// TwinCAT 3 PLC project PLC
// ProgramVersion: 3.1.4023.0
// libraries:
//   Tc2_Standard, * (Beckhoff Automation GmbH)
//   Tc2_System, * (Beckhoff Automation GmbH)
//   Tc3_Module, * (Beckhoff Automation GmbH)
//   VisuSymbols,3.5.10.0,System
// project tree:
//   / GlobalTextList.TcGTLO, PlcTask.TcTTO, Visualization Manager.TcVMO (not stored)
//   GVLs/ Inputs.TcGVL, Outputs.TcGVL, Process.TcGVL
//   POUs/ IIRFilter.TcPOU, UpdateInterlockAndLimit.TcPOU, WriteToInterlockAndLimit.TcPOU, ByteArrayToDINT.TcPOU, ByteArrayToReal.TcPOU, CAN_Receive.TcPOU, CAN_Send.TcPOU, DINTToByteArray.TcPOU, MAIN.TcPOU, RealToByteArray.TcPOU, ScalingIn.TcPOU, ScalingOut.TcPOU
//   VISUs/ Visualization.TcVIS
// real-time tasks:
//   TASK PlcTask: cycle T#2ms, priority 20, ADS port 350
// motion (NC):
//   TASK NC-Task 1 SAF: cycle T#2ms, priority 4, ADS port 501
//   TASK NC-Task 1 SVB: cycle T#2ms, priority 8, ADS port 511
//   AXIS Axis 1 (id 1)
//     OtherSettings: AllowMotionCmdToSlave=true
//     encoder EncType=4
//       EncPara: MaxCount=#x0000ffff
//         Inc: RefSoftSyncMask=#x0000ffff
//     drive DrvType=24
//       Analog: TorqueSetpointScale=10, ScaleFactorActTorque=0.1
//       TimeComp: TaskDelayCycles=1
//     controller CtrType=1
//       CtrPara: PriorControlFactor=1
//         Observer: BandWidth=20
//   AXIS Axis 2 (id 2)
//     OtherSettings: AllowMotionCmdToSlave=true
//     encoder EncType=4
//       EncPara: ScaleFactorNumerator=0.000624, MaxCount=#x0000ffff
//         Inc: RefSoftSyncMask=#x0000ffff
//     drive DrvType=24
//       Analog: TorqueSetpointScale=10, ScaleFactorActTorque=0.1
//       TimeComp: TaskDelayCycles=1
//     controller CtrType=1
//       CtrPara: PriorControlFactor=1
//         Observer: BandWidth=20
//   AXIS Axis 3 (id 3)
//     OtherSettings: AllowMotionCmdToSlave=true
//     encoder EncType=4
//       EncPara: MaxCount=#x0000ffff
//         Inc: RefSoftSyncMask=#x0000ffff
//     drive DrvType=24
//       Analog: TorqueSetpointScale=10, ScaleFactorActTorque=0.1
//       TimeComp: TaskDelayCycles=1
//     controller CtrType=1
//       CtrPara: PriorControlFactor=1
//         Observer: BandWidth=20
//   AXIS Axis 4 (id 4)
//     OtherSettings: AllowMotionCmdToSlave=true
//     encoder EncType=4
//       EncPara: MaxCount=#x0000ffff
//         Inc: RefSoftSyncMask=#x0000ffff
//     drive DrvType=24
//       Analog: TorqueSetpointScale=10, ScaleFactorActTorque=0.1
//       TimeComp: TaskDelayCycles=1
//     controller CtrType=1
//       CtrPara: PriorControlFactor=1
//         Observer: BandWidth=20
// I/O:
//   DEVICE Device 1 (EtherCAT), AmsNetId 5.89.199.32.2.1
//     Term 1 (EK1200) [EK1200-5000 EtherCAT Power supply (2A E-Bus)]
//       Term 2 (EL2008) [EL2008 8Ch. Dig. Output 24V, 0.5A]
//       Term 3 (EL3174) [EL3174 4Ch. Ana. Input +/-10V Diff., +/-20mA SingleEnded, 16 Bit]
//       Term 4 (EL1008) [EL1008 8Ch. Dig. Input 24V, 3ms]
//       Term 6 (EL4132) [EL4132 2Ch. Ana. Output +/-10V, 16bit]
//       Term 7 (EL4132) [EL4132 2Ch. Ana. Output +/-10V, 16bit]
//       Term 8 (EL6751) [EL6751 CANopen Master]
//       Term 9 (EK1110) [EK1110 EtherCAT extension]
//     Term 10 (EK1100) [EK1100 EtherCAT Coupler (2A E-Bus)]
//       Term 11 (EL7031) [EL7031 1Ch. Stepper motor output stage (24V, 1.5A)]
//       Term 12 (EL7031) [EL7031 1Ch. Stepper motor output stage (24V, 1.5A)]
//       Term 13 (EL7031) [EL7031 1Ch. Stepper motor output stage (24V, 1.5A)]
//       Term 14 (EL7031) [EL7031 1Ch. Stepper motor output stage (24V, 1.5A)]
//       Term 15 (EL1008) [EL1008 8Ch. Dig. Input 24V, 3ms]
//       Term 16 (EL3174) [EL3174 4Ch. Ana. Input +/-10V Diff., +/-20mA SingleEnded, 16 Bit]
//       Term 17 (EL3356-0010) [EL3356-0010 1Ch. Ana. Input Resistor Bridge Terminal, 24bit, High Precision]
//       Term 18 (EL3356-0010) [EL3356-0010 1Ch. Ana. Input Resistor Bridge Terminal, 24bit, High Precision]
//       Term 19 (EL3356-0010) [EL3356-0010 1Ch. Ana. Input Resistor Bridge Terminal, 24bit, High Precision]
//       Term 5 (EL4112) [EL4112 2Ch. Ana. Output  0-20mA, 16bit]
//       Term 20 (EL9011) [EL9011 End Terminal]
//   DEVICE Device 2 (EL6751), AmsNetId 5.89.199.32.3.1
//     Box 21 (CAN Interface)
// variable links:
//   NC-Task 1 SAF/Axes/Axis 1 <-> Device 1 (EtherCAT)/Term 10 (EK1100)/Term 11 (EL7031)
//     Drive/Inputs/In/nState1 @bit 3 <-> STM Status/Status/Error
//     Drive/Inputs/In/nState1 @bit 5 <-> STM Status/Status/Moving negative
//     Drive/Inputs/In/nState1 @bit 4 <-> STM Status/Status/Moving positive
//     Drive/Inputs/In/nState1 @bit 1 <-> STM Status/Status/Ready
//     Drive/Inputs/In/nState1 <-> STM Status/Status/Ready to enable
//     Drive/Inputs/In/nState1 @bit 6 <-> STM Status/Status/Torque reduced
//     Drive/Inputs/In/nState1 @bit 2 <-> STM Status/Status/Warning
//     Drive/Inputs/In/nState2 @bit 3 <-> STM Status/Status/Digital input 1
//     Drive/Inputs/In/nState2 @bit 4 <-> STM Status/Status/Digital input 2
//     Drive/Inputs/In/nState2 @bit 5 <-> STM Status/Status/Sync error
//     Drive/Inputs/In/nState2 @bit 7 <-> STM Status/Status/TxPDO Toggle
//     Drive/Inputs/In/nState4 @bit 1 <-> WcState/InputToggle
//     Drive/Inputs/In/nState4 <-> WcState/WcState
//     Drive/Outputs/Out/nCtrl1 <-> STM Control/Control/Enable
//     Drive/Outputs/Out/nCtrl1 @bit 2 <-> STM Control/Control/Reduce torque
//     Drive/Outputs/Out/nCtrl1 @bit 1 <-> STM Control/Control/Reset
//     Drive/Outputs/Out/nDataOut2[0] <-> STM Velocity/Velocity
//     Enc/Inputs/In/nDataIn1[0] <-> ENC Status compact/Counter value
//     Enc/Inputs/In/nDataIn2[0] <-> ENC Status compact/Latch value
//     Enc/Inputs/In/nState1 @bit 4 <-> ENC Status compact/Status/Counter overflow
//     Enc/Inputs/In/nState1 @bit 3 <-> ENC Status compact/Status/Counter underflow
//     Enc/Inputs/In/nState1 @bit 1 <-> ENC Status compact/Status/Latch extern valid
//     Enc/Inputs/In/nState1 @bit 2 <-> ENC Status compact/Status/Set counter done
//     Enc/Inputs/In/nState2 @bit 4 <-> ENC Status compact/Status/Status of extern latch
//     Enc/Inputs/In/nState2 @bit 5 <-> ENC Status compact/Status/Sync error
//     Enc/Inputs/In/nState2 @bit 7 <-> ENC Status compact/Status/TxPDO Toggle
//     Enc/Inputs/In/nState4 @bit 1 <-> WcState/InputToggle
//     Enc/Inputs/In/nState4 <-> WcState/WcState
//     Enc/Outputs/Out/nCtrl1 @bit 3 <-> ENC Control compact/Control/Enable latch extern on negative edge
//     Enc/Outputs/Out/nCtrl1 @bit 1 <-> ENC Control compact/Control/Enable latch extern on positive edge
//     Enc/Outputs/Out/nCtrl1 @bit 2 <-> ENC Control compact/Control/Set counter
//     Enc/Outputs/Out/nDataOut1[0] <-> ENC Control compact/Set counter value
//   NC-Task 1 SAF/Axes/Axis 2 <-> Device 1 (EtherCAT)/Term 10 (EK1100)/Term 12 (EL7031)
//     Drive/Inputs/In/nState1 @bit 3 <-> STM Status/Status/Error
//     Drive/Inputs/In/nState1 @bit 5 <-> STM Status/Status/Moving negative
//     Drive/Inputs/In/nState1 @bit 4 <-> STM Status/Status/Moving positive
//     Drive/Inputs/In/nState1 @bit 1 <-> STM Status/Status/Ready
//     Drive/Inputs/In/nState1 <-> STM Status/Status/Ready to enable
//     Drive/Inputs/In/nState1 @bit 6 <-> STM Status/Status/Torque reduced
//     Drive/Inputs/In/nState1 @bit 2 <-> STM Status/Status/Warning
//     Drive/Inputs/In/nState2 @bit 3 <-> STM Status/Status/Digital input 1
//     Drive/Inputs/In/nState2 @bit 4 <-> STM Status/Status/Digital input 2
//     Drive/Inputs/In/nState2 @bit 5 <-> STM Status/Status/Sync error
//     Drive/Inputs/In/nState2 @bit 7 <-> STM Status/Status/TxPDO Toggle
//     Drive/Inputs/In/nState4 @bit 1 <-> WcState/InputToggle
//     Drive/Inputs/In/nState4 <-> WcState/WcState
//     Drive/Outputs/Out/nCtrl1 <-> STM Control/Control/Enable
//     Drive/Outputs/Out/nCtrl1 @bit 2 <-> STM Control/Control/Reduce torque
//     Drive/Outputs/Out/nCtrl1 @bit 1 <-> STM Control/Control/Reset
//     Drive/Outputs/Out/nDataOut2[0] <-> STM Velocity/Velocity
//     Enc/Inputs/In/nDataIn1[0] <-> ENC Status compact/Counter value
//     Enc/Inputs/In/nDataIn2[0] <-> ENC Status compact/Latch value
//     Enc/Inputs/In/nState1 @bit 4 <-> ENC Status compact/Status/Counter overflow
//     Enc/Inputs/In/nState1 @bit 3 <-> ENC Status compact/Status/Counter underflow
//     Enc/Inputs/In/nState1 @bit 1 <-> ENC Status compact/Status/Latch extern valid
//     Enc/Inputs/In/nState1 @bit 2 <-> ENC Status compact/Status/Set counter done
//     Enc/Inputs/In/nState2 @bit 4 <-> ENC Status compact/Status/Status of extern latch
//     Enc/Inputs/In/nState2 @bit 5 <-> ENC Status compact/Status/Sync error
//     Enc/Inputs/In/nState2 @bit 7 <-> ENC Status compact/Status/TxPDO Toggle
//     Enc/Inputs/In/nState4 @bit 1 <-> WcState/InputToggle
//     Enc/Inputs/In/nState4 <-> WcState/WcState
//     Enc/Outputs/Out/nCtrl1 @bit 3 <-> ENC Control compact/Control/Enable latch extern on negative edge
//     Enc/Outputs/Out/nCtrl1 @bit 1 <-> ENC Control compact/Control/Enable latch extern on positive edge
//     Enc/Outputs/Out/nCtrl1 @bit 2 <-> ENC Control compact/Control/Set counter
//     Enc/Outputs/Out/nDataOut1[0] <-> ENC Control compact/Set counter value
//   NC-Task 1 SAF/Axes/Axis 3 <-> Device 1 (EtherCAT)/Term 10 (EK1100)/Term 13 (EL7031)
//     Drive/Inputs/In/nState1 @bit 3 <-> STM Status/Status/Error
//     Drive/Inputs/In/nState1 @bit 5 <-> STM Status/Status/Moving negative
//     Drive/Inputs/In/nState1 @bit 4 <-> STM Status/Status/Moving positive
//     Drive/Inputs/In/nState1 @bit 1 <-> STM Status/Status/Ready
//     Drive/Inputs/In/nState1 <-> STM Status/Status/Ready to enable
//     Drive/Inputs/In/nState1 @bit 6 <-> STM Status/Status/Torque reduced
//     Drive/Inputs/In/nState1 @bit 2 <-> STM Status/Status/Warning
//     Drive/Inputs/In/nState2 @bit 3 <-> STM Status/Status/Digital input 1
//     Drive/Inputs/In/nState2 @bit 4 <-> STM Status/Status/Digital input 2
//     Drive/Inputs/In/nState2 @bit 5 <-> STM Status/Status/Sync error
//     Drive/Inputs/In/nState2 @bit 7 <-> STM Status/Status/TxPDO Toggle
//     Drive/Inputs/In/nState4 @bit 1 <-> WcState/InputToggle
//     Drive/Inputs/In/nState4 <-> WcState/WcState
//     Drive/Outputs/Out/nCtrl1 <-> STM Control/Control/Enable
//     Drive/Outputs/Out/nCtrl1 @bit 2 <-> STM Control/Control/Reduce torque
//     Drive/Outputs/Out/nCtrl1 @bit 1 <-> STM Control/Control/Reset
//     Drive/Outputs/Out/nDataOut2[0] <-> STM Velocity/Velocity
//     Enc/Inputs/In/nDataIn1[0] <-> ENC Status compact/Counter value
//     Enc/Inputs/In/nDataIn2[0] <-> ENC Status compact/Latch value
//     Enc/Inputs/In/nState1 @bit 4 <-> ENC Status compact/Status/Counter overflow
//     Enc/Inputs/In/nState1 @bit 3 <-> ENC Status compact/Status/Counter underflow
//     Enc/Inputs/In/nState1 @bit 1 <-> ENC Status compact/Status/Latch extern valid
//     Enc/Inputs/In/nState1 @bit 2 <-> ENC Status compact/Status/Set counter done
//     Enc/Inputs/In/nState2 @bit 4 <-> ENC Status compact/Status/Status of extern latch
//     Enc/Inputs/In/nState2 @bit 5 <-> ENC Status compact/Status/Sync error
//     Enc/Inputs/In/nState2 @bit 7 <-> ENC Status compact/Status/TxPDO Toggle
//     Enc/Inputs/In/nState4 @bit 1 <-> WcState/InputToggle
//     Enc/Inputs/In/nState4 <-> WcState/WcState
//     Enc/Outputs/Out/nCtrl1 @bit 3 <-> ENC Control compact/Control/Enable latch extern on negative edge
//     Enc/Outputs/Out/nCtrl1 @bit 1 <-> ENC Control compact/Control/Enable latch extern on positive edge
//     Enc/Outputs/Out/nCtrl1 @bit 2 <-> ENC Control compact/Control/Set counter
//     Enc/Outputs/Out/nDataOut1[0] <-> ENC Control compact/Set counter value
//   NC-Task 1 SAF/Axes/Axis 4 <-> Device 1 (EtherCAT)/Term 10 (EK1100)/Term 14 (EL7031)
//     Drive/Inputs/In/nState1 @bit 3 <-> STM Status/Status/Error
//     Drive/Inputs/In/nState1 @bit 5 <-> STM Status/Status/Moving negative
//     Drive/Inputs/In/nState1 @bit 4 <-> STM Status/Status/Moving positive
//     Drive/Inputs/In/nState1 @bit 1 <-> STM Status/Status/Ready
//     Drive/Inputs/In/nState1 <-> STM Status/Status/Ready to enable
//     Drive/Inputs/In/nState1 @bit 6 <-> STM Status/Status/Torque reduced
//     Drive/Inputs/In/nState1 @bit 2 <-> STM Status/Status/Warning
//     Drive/Inputs/In/nState2 @bit 3 <-> STM Status/Status/Digital input 1
//     Drive/Inputs/In/nState2 @bit 4 <-> STM Status/Status/Digital input 2
//     Drive/Inputs/In/nState2 @bit 5 <-> STM Status/Status/Sync error
//     Drive/Inputs/In/nState2 @bit 7 <-> STM Status/Status/TxPDO Toggle
//     Drive/Inputs/In/nState4 @bit 1 <-> WcState/InputToggle
//     Drive/Inputs/In/nState4 <-> WcState/WcState
//     Drive/Outputs/Out/nCtrl1 <-> STM Control/Control/Enable
//     Drive/Outputs/Out/nCtrl1 @bit 2 <-> STM Control/Control/Reduce torque
//     Drive/Outputs/Out/nCtrl1 @bit 1 <-> STM Control/Control/Reset
//     Drive/Outputs/Out/nDataOut2[0] <-> STM Velocity/Velocity
//     Enc/Inputs/In/nDataIn1[0] <-> ENC Status compact/Counter value
//     Enc/Inputs/In/nDataIn2[0] <-> ENC Status compact/Latch value
//     Enc/Inputs/In/nState1 @bit 4 <-> ENC Status compact/Status/Counter overflow
//     Enc/Inputs/In/nState1 @bit 3 <-> ENC Status compact/Status/Counter underflow
//     Enc/Inputs/In/nState1 @bit 1 <-> ENC Status compact/Status/Latch extern valid
//     Enc/Inputs/In/nState1 @bit 2 <-> ENC Status compact/Status/Set counter done
//     Enc/Inputs/In/nState2 @bit 4 <-> ENC Status compact/Status/Status of extern latch
//     Enc/Inputs/In/nState2 @bit 5 <-> ENC Status compact/Status/Sync error
//     Enc/Inputs/In/nState2 @bit 7 <-> ENC Status compact/Status/TxPDO Toggle
//     Enc/Inputs/In/nState4 @bit 1 <-> WcState/InputToggle
//     Enc/Inputs/In/nState4 <-> WcState/WcState
//     Enc/Outputs/Out/nCtrl1 @bit 3 <-> ENC Control compact/Control/Enable latch extern on negative edge
//     Enc/Outputs/Out/nCtrl1 @bit 1 <-> ENC Control compact/Control/Enable latch extern on positive edge
//     Enc/Outputs/Out/nCtrl1 @bit 2 <-> ENC Control compact/Control/Set counter
//     Enc/Outputs/Out/nDataOut1[0] <-> ENC Control compact/Set counter value
//   PLC/PLC Instance <-> Device 1 (EtherCAT)/Term 1 (EK1200)/Term 2 (EL2008)
//     PlcTask Outputs/Outputs.DO_PumpEnable <-> Channel 8/Output
//     PlcTask Outputs/Outputs.bool1 <-> Channel 4/Output
//     PlcTask Outputs/Outputs.bool2 <-> Channel 5/Output
//     PlcTask Outputs/Outputs.bool3 <-> Channel 6/Output
//   PLC/PLC Instance <-> Device 1 (EtherCAT)/Term 1 (EK1200)/Term 7 (EL4132)
//     PlcTask Outputs/Outputs.AO_HOISTING <-> Channel 1/Output
//     PlcTask Outputs/Outputs.AO_PUMP <-> Channel 2/Output
//   PLC/PLC Instance <-> Device 1 (EtherCAT)/Term 10 (EK1100)/Term 15 (EL1008)
//     PlcTask Inputs/Inputs.DI_HOISTING_LIM_BOTTOM <-> Channel 6/Input
//     PlcTask Inputs/Inputs.DI_HOISTING_LIM_TOP <-> Channel 5/Input
//     PlcTask Inputs/Inputs.DI_STABLIZER_LIM_HOIST_SIDE <-> Channel 2/Input
//     PlcTask Inputs/Inputs.DI_STABLIZER_LIM_OPPOSITE_HOIST <-> Channel 4/Input
//     PlcTask Inputs/Inputs.DOORSENS1 <-> Channel 1/Input
//     PlcTask Inputs/Inputs.DOORSENS2 <-> Channel 3/Input
//   PLC/PLC Instance <-> Device 1 (EtherCAT)/Term 10 (EK1100)/Term 16 (EL3174)
//     PlcTask Inputs/Inputs.AI_HEIGHT <-> AI Standard Channel 3/Value
//     PlcTask Inputs/Inputs.AI_PressureSensor <-> AI Standard Channel 2/Value
//     PlcTask Inputs/Inputs.AI_TEMP <-> AI Standard Channel 1/Value
//   PLC/PLC Instance <-> Device 1 (EtherCAT)/Term 10 (EK1100)/Term 17 (EL3356-0010)
//     PlcTask Inputs/Inputs.AI_Z1 <-> RMB Value (Real)/Value (Real)
//   PLC/PLC Instance <-> Device 1 (EtherCAT)/Term 10 (EK1100)/Term 18 (EL3356-0010)
//     PlcTask Inputs/Inputs.AI_Z2 <-> RMB Value (Real)/Value (Real)
//   PLC/PLC Instance <-> Device 1 (EtherCAT)/Term 10 (EK1100)/Term 19 (EL3356-0010)
//     PlcTask Inputs/Inputs.AI_Z3 <-> RMB Value (Real)/Value (Real)
//   PLC/PLC Instance <-> Device 1 (EtherCAT)/Term 10 (EK1100)/Term 5 (EL4112)
//     PlcTask Outputs/Outputs.AO_ValveWaterIn <-> Channel 1/Output
//   PLC/PLC Instance <-> Device 2 (EL6751)/Box 21 (CAN Interface)
//     PlcTask Inputs/Inputs.RxQueue <-> Inputs/RxQueue
//     PlcTask Outputs/Outputs.TxQueue <-> Outputs/TxQueue

CONFIGURATION PLC
    RESOURCE PLC ON TwinCAT3
        TASK PlcTask(INTERVAL := T#2ms, PRIORITY := 20);
        PROGRAM MAIN WITH PlcTask : MAIN;
    END_RESOURCE
END_CONFIGURATION

// ---- GVLs/Inputs.TcGVL
{attribute 'qualified_only'}
VAR_GLOBAL
	// INTERLOCK
	DOORSENS1 AT %I* : BOOL;
	DOORSENS2 AT %I* : BOOL;
	
	// ANALOG IN
	AI_PressureSensor AT %I* :UINT;
	AI_RPM AT %I* : UINT;
	AI_TORQUE AT %I* : UINT;
	AI_Z1 AT %I* : REAL;
	AI_Z2 AT %I* : REAL;
	AI_Z3 AT %I* : REAL;
	AI_TEMP AT %I* : UINT;
	AI_HEIGHT AT %I* : UINT;
	AI_WaterInPressure AT %I*: UINT;

	
	
	// DIGITAL IN
	DI_HOISTING_LIM_TOP AT %I*: BOOL;
	DI_HOISTING_LIM_BOTTOM AT %I*: BOOL;
	
	DI_STABLIZER_LIM_HOIST_SIDE AT %I*: BOOL;
	DI_STABLIZER_LIM_OPPOSITE_HOIST AT %I*: BOOL;
	
	// CAN-BUS
	//TxCounter AT %I* : UINT;
	//RxCounter AT %I* : UINT;
	//NoOfRxMessages AT %I* : UINT;
	//RxMessages AT %I* : ARRAY [0..99] OF CANQUEUE;
	
	RxQueue AT %I*: CANRXQUEUESTRUCT_N_100;
	
	
END_VAR

// ---- GVLs/Outputs.TcGVL
{attribute 'qualified_only'}
VAR_GLOBAL
	
	// ANALOG OUT
	AO_RPM AT %Q* : INT;
	AO_TORQUE AT %Q* : INT;
	AO_HOISTING AT %Q* : INT;
	AO_PUMP AT %Q* : INT;
	AO_ValveWaterIn AT %Q* : INT;
	
	
	DO_PumpEnable AT %Q*: BOOL;
	// CAN
	TxQueue AT %Q* : CANTXQUEUESTRUCT_N_100;
	
	bool1 AT %Q* : BOOL;
	bool2 AT %Q* : BOOL;
	bool3 AT %Q* : BOOL;
	
END_VAR

// ---- GVLs/Process.TcGVL
{attribute 'qualified_only'}
VAR_GLOBAL
	// INPUTS
	State : DINT := 0;
	Pressure: REAL;
	Temperature: REAL;
	InterlockAndLimit: DINT := 127;
	TopDriveRPM : REAL := 465.2;
	TopDriveTorque : REAL := 34.4;
	WOB_1 : REAL := 12.3;
	WOB_2 : REAL := 12.3;
	WOB_3 : REAL := 12.3;
	WOB_AVG : REAL := (WOB_1 + WOB_2 + WOB_3)/3;
	Height : REAL;
	CurrentHeight : REAL;
	
	// OUTPUTS
	TopDriveRPMSetPoint : REAL := 465.0;
	TopDriveTorqueSetPoint : REAL := 34.0;
	PumpSetPoint: REAL := 50.0;
	HoistingSpeed: REAL;
	//HoistingEnable: BOOL := FALSE;
	
	
	// GUI inputs
	HoistingEnable : DINT;
	HoistingDemandValue: REAL;
	
	PumpEnable : DINT;
	PumpOpen : DINT;
	PumpPID: REAL;
	
	TopDriveEnable : DINT;
	InputTopDriveRPMSetPoint : REAL;
	InputTopDriveTorqueSetPoint : REAL;
	
END_VAR

// ---- POUs/MAIN.TcPOU
PROGRAM MAIN
VAR
	startup : BOOL := TRUE;
END_VAR

CAN_Receive();
ScalingIn();

Outputs.bool1 := DINT_TO_BOOL(Process.HoistingEnable);
Outputs.bool2 := DINT_TO_BOOL(Process.HoistingEnable);
Outputs.bool3 := DINT_TO_BOOL(Process.HoistingEnable);

CASE Process.State OF
	0:
		Process.HoistingDemandValue := 100;
		IF NOT Inputs.DI_HOISTING_LIM_TOP THEN
			Process.State := 1;
			Process.HoistingDemandValue := 0;
		END_IF
	
END_CASE

UpdateInterlockAndLimit();
ScalingOut();
CAN_Send();

END_PROGRAM

// ---- POUs/CAN_Receive.TcPOU
FUNCTION CAN_Receive : BOOL
VAR_INPUT
END_VAR
VAR
	// CAN-BUS
	arrCobId : ARRAY [0..45]OF UINT;
	arrCobIdTmp : ARRAY [0..45]OF UINT;
	MessageReceived: ARRAY [0..9] OF CANQUEUE;
	test_number_1 : REAL;
	test_number_2 : REAL;
	test : CANQUEUE;
	MsgId : UINT;
	// Indexing vars
	i: UINT;
	j : UINT;

	z: UINT;
	n: INT;
	z_old: UINT;
END_VAR

(* Receiving, CAN-BUS *)
IF Outputs.TxQueue.RxCounter <> Inputs.RxQueue.RxCounter THEN
	FOR i := 0 TO (Inputs.RxQueue.NoOfRxMessages-1) DO
		MessageReceived[i] := Inputs.RxQueue.RxMessages[i];
	END_FOR
	Outputs.TxQueue.RxCounter := Outputs.TxQueue.RxCounter+1;
END_IF

(*
IF (Inputs.NoOfRxMessages = 0) THEN
	RETURN;
END_IF
*)


(*Parsing*)
FOR z:=0 TO (Inputs.RxQueue.NoOfRxMessages) DO
	 (*Logging last 45 received CobId's*)
	IF z<>z_old AND n<45 THEN
		arrCobId[n]:=MessageReceived[z].cobId;
		IF n>=44 THEN n:=0;arrCobIdTmp:=arrCobId; ELSE n:=n+1; END_IF
		z_old:=z;
	END_IF
	
	//Removes the last five bits in number and shifts five places
	MsgId := SHR(MessageReceived[z].cobId AND 16#FFE0, 5);

	(*Case structure to catch specific CobId and parse data from it*)
	CASE  MsgId OF		
			
		40: (* Engine Oil Pressure *)
			test := MessageReceived[z];
			
		//ELSE // DEBUG
		//	J1939_UNKNOWN_COBID	:=MessageReceived[z];
		//	J1939_createVisString(rxData:=ADR(MessageReceived[z].rxData) , strRxData=>strJ1939_UNKNOWN_COBID );
			// DISPLAY UNKNOW MESSAGES
	//		ADSLOGSTR(msgCtrlMask:=ADSLOG_MSGTYPE_HINT , msgFmtStr:= 'J1939 uknown CobId: ' , strArg:=strJ1939_UNKNOWN_COBID );
	
		200:
			ByteArrayToReal(MessageReceived[z],0, output => test_number_1);
			ByteArrayToReal(MessageReceived[z],4, output => test_number_2);
		
		201:
			ByteArrayToDINT(MessageReceived[z], 0, output => Process.PumpOpen);
			
		202:
			ByteArrayToDINT(MessageReceived[z], 0, output => Process.HoistingEnable);
			ByteArrayToReal(MessageReceived[z], 4, output => Process.HoistingDemandValue);
			
		203:
			ByteArrayToDINT(MessageReceived[z], 0, output => Process.PumpEnable);
			ByteArrayToReal(MessageReceived[z], 4, output => Process.PumpPID);
			
		206:
			ByteArrayToReal(MessageReceived[z], 0, output => Process.InputTopDriveRPMSetPoint);
			ByteArrayToReal(MessageReceived[z], 4, output => Process.InputTopDriveTorqueSetPoint);
			
		208:
			ByteArrayToDINT(MessageReceived[z], 0, output => Process.TopDriveEnable);
	END_CASE
END_FOR

END_FUNCTION

// ---- POUs/ByteArrayToReal.TcPOU
FUNCTION ByteArrayToReal : REAL
VAR_INPUT
	msg : CANQUEUE;
	pos : INT;
END_VAR
VAR_OUTPUT
	output : REAL;
END_VAR
VAR
	tmp: ARRAY[0..3] OF USINT;
	pt : POINTER TO REAL;
	i : INT;
END_VAR

FOR i := 0 TO 3 DO
	tmp[i] := msg.data[i+pos];
END_FOR
pt := ADR(tmp);
output := pt^;

END_FUNCTION

// ---- POUs/ByteArrayToDINT.TcPOU
FUNCTION ByteArrayToDINT : DINT
VAR_INPUT
	msg : CANQUEUE;
	pos : INT;
END_VAR
VAR_OUTPUT
	output : DINT;
END_VAR
VAR
	result : UDINT;
	i: INT;
END_VAR

FOR i := pos + 3 TO 0 BY -1 DO
	// starts with the last number in the array and shifts it zero places
	// the following numbers get shiftet left one more place than the last and added to the total.
	result := result + (SHL(USINT_TO_UDINT(msg.data[i]), (3-i)* 8));
END_FOR
output := UDINT_TO_DINT(result);

END_FUNCTION

// ---- POUs/ScalingIn.TcPOU
FUNCTION ScalingIn : BOOL
VAR_INPUT
END_VAR
VAR
END_VAR

Process.currentHeight:= Inputs.AI_HEIGHT*(0.0263) + 79.878;
IIRFilter(Process.currentHeight,0.99,Process.Height);
//Process.Height := Inputs.AI_HEIGHT*(-0.00508825) + 49.10937731;

// Circulation system pressure
Process.Pressure := Inputs.AI_PressureSensor*0.003277 - 0.12124;

// Circluation system temperature
Process.Temperature := Inputs.AI_TEMP*0.003282 - 0.1083;

END_FUNCTION

// ---- POUs/IIRFilter.TcPOU
FUNCTION IIRFilter : REAL
VAR_INPUT
	newValue : REAL;
	filterStrength : REAL;
END_VAR
VAR_IN_OUT
	value : REAL;
END_VAR
VAR
END_VAR

value := newValue*(1-filterStrength) + value*filterStrength;

END_FUNCTION

// ---- POUs/UpdateInterlockAndLimit.TcPOU
FUNCTION UpdateInterlockAndLimit
VAR_INPUT
END_VAR
VAR
END_VAR

//Resets the interlock to allow for 
Process.InterlockAndLimit := 0;
WriteToInterlockAndLimit(Inputs.DOORSENS1,0);
WriteToInterlockAndLimit(Inputs.DOORSENS2,1);
WriteToInterlockAndLimit(Inputs.DI_HOISTING_LIM_BOTTOM,2);
WriteToInterlockAndLimit(Inputs.DI_HOISTING_LIM_TOP,3);
WriteToInterlockAndLimit(Inputs.DI_STABLIZER_LIM_HOIST_SIDE,4);
WriteToInterlockAndLimit(Inputs.DI_STABLIZER_LIM_OPPOSITE_HOIST,5);

END_FUNCTION

// ---- POUs/WriteToInterlockAndLimit.TcPOU
FUNCTION WriteToInterlockAndLimit
VAR_INPUT
	value: BOOL;
	pos: DINT;
END_VAR
VAR
	BoolNumber : UDINT;
	result : UDINT;
END_VAR

BoolNumber := SHL(BOOL_TO_UDINT(value AND 1),pos);
result := DINT_TO_UDINT(Process.InterlockAndLimit) OR BoolNumber;
Process.InterlockAndLimit := UDINT_TO_DINT(result);

END_FUNCTION

// ---- POUs/ScalingOut.TcPOU
FUNCTION ScalingOut : BOOL
VAR_INPUT
END_VAR
VAR
	HoistingScaling: INT := 300;
	PumpScaling: INT := 100;
	IntMax : INT := 32767;
END_VAR

//Allows no motor movement when either door is open
IF (Inputs.DOORSENS1 = FALSE OR Inputs.DOORSENS2 = FALSE) THEN
	Outputs.AO_HOISTING := 0;
	RETURN;
END_IF

// Prevent integer overflow which causes motor to run in reverse
IF Process.HoistingDemandValue >= HoistingScaling THEN
	Process.HoistingDemandValue := INT_TO_REAL(HoistingScaling);
ELSIF Process.HoistingDemandValue <= (-1) * HoistingScaling THEN
	Process.HoistingDemandValue:= INT_TO_REAL(HoistingScaling*(-1));
END_IF

//Prevent integer overflow and sub-zero values
IF Process.PumpPID >= PumpScaling THEN
	Process.PumpPID := REAL_TO_INT(PumpScaling);
ELSIF Process.PumpPID <= 0 THEN
	Process.PumpPID := 0;
END_IF


//Only downwards when top switch is pressed
IF (Inputs.DI_HOISTING_LIM_TOP = FALSE) AND (Process.HoistingDemandValue > 0) THEN
	Outputs.AO_HOISTING := 0;
//Only upwards when bottom switch is pressed
ELSIF (Inputs.DI_HOISTING_LIM_BOTTOM = FALSE) AND (Process.HoistingDemandValue < 0) THEN
	Outputs.AO_HOISTING := 0;
ELSE
	Outputs.AO_HOISTING := REAL_TO_INT(Process.HoistingDemandValue/HoistingScaling*IntMax);
END_IF

Outputs.AO_ValveWaterIn := DINT_TO_INT(Process.PumpOpen*IntMax);

Outputs.DO_PumpEnable := DINT_TO_BOOL(Process.PumpEnable);
Outputs.AO_PUMP := REAL_TO_INT(Process.PumpPID/PumpScaling*IntMax);

END_FUNCTION

// ---- POUs/CAN_Send.TcPOU
FUNCTION CAN_Send : BOOL
VAR_INPUT
END_VAR
VAR
	NumberOfMessagesToSend : UINT := 9;
	MessageToSend : ARRAY [0..9] OF CANQUEUE;
	// msg

	
	k : UINT;
END_VAR

//System State, ID 100
MessageToSend[0].cobId :=  SHL(100, 5) OR 8;
DINTToByteArray(Process.State, 0, msg => MessageToSend[0].data);

//WOB_1 and WOB_2, ID 110
MessageToSend[1].cobId := SHL(110, 5) OR 8;
REALToByteArray(Inputs.AI_Z1,Inputs.AI_Z2, msg => MessageToSend[1].data);

//WOB_3 and WOB_AVG, ID 120
MessageToSend[2].cobId :=  SHL(120, 5) OR 8;
REALToByteArray(Inputs.AI_Z3, Inputs.AI_Z1+Inputs.AI_Z2+Inputs.AI_Z3, msg => MessageToSend[2].data);

//Pressure and temperature (circulation sysstem), ID 130
MessageToSend[3].cobId :=  SHL(130, 5) OR 8;
RealToByteArray(Process.Pressure, Process.Temperature, msg => MessageToSend[3].data);

//Interlocks, ID 140
MessageToSend[4].cobId := SHL(140, 5) OR 8;
DINTToByteArray(Process.InterlockAndLimit,0, msg => MessageToSend[4].data);

//Pump set point, ID 150
MessageToSend[5].cobId := SHL(150, 5) OR 8;
REALToByteArray(Process.PumpSetPoint,Process.Height, msg => MessageToSend[5].data);

//Top drive RPM and Torque, ID 160
MessageToSend[6].cobId :=  SHL(160, 5) OR 8;
RealToByteArray(Process.TopDriveRPM, Process.TopDriveTorque, msg => MessageToSend[6].data);

//Set point top drive RPM and torque, ID 170
MessageToSend[7].cobId := SHL(170, 5) OR 8;
REALToByteArray(Process.TopDriveRPMSetPoint,Process.TopDriveTorqueSetPoint, msg => MessageToSend[7].data);

//Signals last message in iteration, ID 199, should always be last in array.
MessageToSend[8].cobId := SHL(199,5) OR 8;



IF Outputs.TxQueue.TxCounter = Inputs.RxQueue.TxCounter THEN
	FOR k:=0 TO NumberOfMessagesToSend DO
		Outputs.TxQueue.TxMessages[k] := MessageToSend[k];
	END_FOR
	Outputs.TxQueue.NoOfTxMessages := NumberOfMessagesToSend;
	Outputs.TxQueue.TxCounter := Outputs.TxQueue.TxCounter +1;
END_IF
k := 0;

END_FUNCTION

// ---- POUs/DINTToByteArray.TcPOU
FUNCTION DINTToByteArray
VAR_OUTPUT
	msg : ARRAY[0..7] OF USINT;
END_VAR
VAR_INPUT
	value1 : DINT;
	value2 : DINT;
END_VAR
VAR
	i : INT;
	temp : UDINT;
END_VAR

//converts two numbers to a byte-array and returns the array
temp := DINT_TO_UDINT(value1);
FOR i := 3 TO 0 BY -1 DO
	msg[i] := UDINT_TO_USINT(temp MOD 256);
	temp := temp / 256;
END_FOR;


temp := DINT_TO_UDINT(value2);
FOR i := 7 TO 4 BY -1 DO
	msg[i] := UDINT_TO_USINT(temp MOD 256);
	temp := temp / 256;
END_FOR;

END_FUNCTION

// ---- POUs/RealToByteArray.TcPOU
FUNCTION RealToByteArray
VAR_OUTPUT
	msg : ARRAY[0..7] OF USINT;
END_VAR
VAR_INPUT
	value1 : REAL;
	value2 : REAL;
END_VAR
VAR
	pt1 : POINTER TO ARRAY[0..3] OF USINT;
	pt2 : POINTER TO ARRAY[0..3] OF USINT;
	i : INT;
END_VAR

//converts two floating point numbers to a byte-array and returns the array.

pt1 := ADR(value1);
pt2 := ADR(value2);
FOR i:=0 TO 3 DO
	msg[i] := pt1^[i];
	msg[i+4] := pt2^[i];
END_FOR;

END_FUNCTION

// ---- VISUs/Visualization.TcVIS
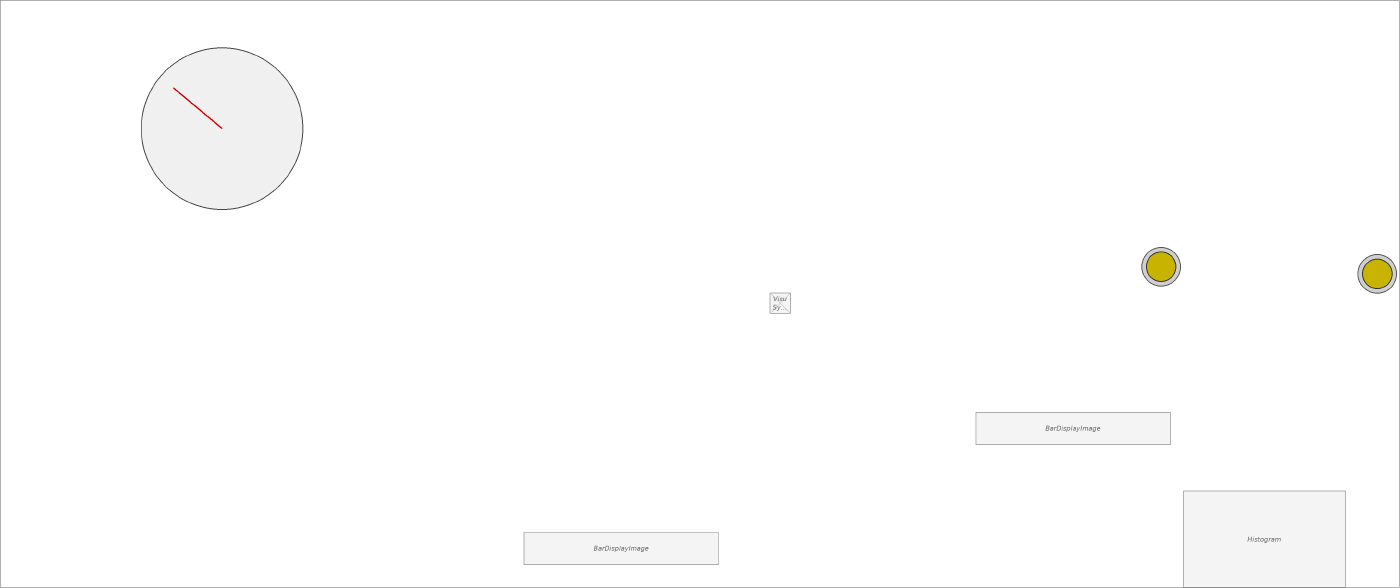
VISUALIZATION Visualization  // 2157x906
    Lamp1 (2087,387 70x70), style: Lamp-Lamp1-Yellow
    Lamp1 (1754,376 70x70), variable: Inputs.DI_HOISTING_LIM_TOP, style: Lamp-Lamp1-Yellow
    Meter360 (217,73 250x250), value: Inputs.AI_PressureSensor, style: Meter-Meter360-Gray, scale format: %.1f, scale 0..100
    BarDisplayImage (807,820 300x50), value: Process.Pressure, style: BarDisplayImage-Gray, scale format: %.1f, scale 0..100
    Histogram (1823,756 250x150), scale format: %.1f, scale 0..100
    BarDisplayImage (1503,635 300x50), value: Process.Temperature, style: BarDisplayImage-Gray, scale format: %.1f, scale 0..100
    Image (1186,451 32x32), text variable: Process.Temperature, image: VisuSymbols.Symbols.Text
END_VISUALIZATION
